{attribute 'linkalways'} 
{attribute 'no_explicit_call' := 'This FB is a CLASS and must be accessed using methods or properties'}
{attribute 'enable_dynamic_creation'}
FUNCTION_BLOCK FINAL SUB_ULINT EXTENDS Node
VAR
	in1 : _ULINT(0);
	in2 : _ULINT(0);
	out : _ULINT(0);
END_VAR

METHOD PUBLIC Clone : I_Node
VAR
	pNode : POINTER TO SUB_ULINT;
END_VAR
pNode := __NEW(SUB_ULINT);
Clone := pNode^;
END_METHOD

METHOD FB_init : BOOL
VAR_INPUT
	bInitRetains : BOOL; // if TRUE, the retain variables are initialized (warm start / cold start)
	bInCopyCode : BOOL;  // if TRUE, the instance afterwards gets moved into the copy code (online change)
END_VAR
AddInput('in1',THIS^.in1);
AddInput('in2',THIS^.in2);
AddOutput('out', THIS^.out);
END_METHOD

METHOD PROTECTED OnExecute
VAR
END_VAR
out.Value := in1.Value - in2.Value;
END_METHOD

END_FUNCTION_BLOCK

(* stored: Version 1.1.0.1, ProductVersion 3.1.4024.15
   POU SUB_ULINT: Id {f241346e-e4fb-48e0-865e-172378182018}, SpecialFunc None
   Folder Constructor: Id {f60f44e9-af4e-40c0-b3fd-18fbc32146f1}
   Method Clone: Id {0de03363-a750-4e72-ab5e-a004e8a8ced2}
   Method FB_init: Id {f34c83b9-f1fe-4b36-8948-f8cd5f93f641}
   Method OnExecute: Id {a19d287b-381f-4b15-8d0b-ed50a5c8d8bc} *)
